PROGRAM MAIN
VAR
	
END_VAR

POU_TestBase();

//AlarmWithCustomSourceInfo();
//OtherAlarmsWithCustomSource();
P_AlarmHandling();
P_AlarmTable();
MultipleAlarmCreation();

P_EventLogger_TCSAlarms();

END_PROGRAM

(* stored: Version 1.1.0.1, ProductVersion 3.1.4024.11
   POU MAIN: Id {1504ce68-47a1-4b47-8617-25bedc0a150a}, SpecialFunc None *)
